FUNCTION_BLOCK EL3014
VAR
	_io : EL3xx4_Data;
	{attribute addProperty Name "WcState"}
	_wcState : WcStateInputToggle;
	{attribute addProperty Name "Info data"}
	_infoData : InfoDataAds;
END_VAR

PROPERTY IO : REFERENCE TO EL3xx4_Data
GET
IO REF= _io;
END_GET
END_PROPERTY

PROPERTY WcState : REFERENCE TO WcStateInputToggle
GET
WcState REF= _wcState;
END_GET
END_PROPERTY

END_FUNCTION_BLOCK

(* stored: Version 1.1.0.1, ProductVersion 3.1.4024.9
   POU EL3014: Id {15204826-2c94-02ae-383a-80dd5a00157f}, SpecialFunc None
   Property IO: Id {5d69b753-5e9f-0a8a-1825-ed3196d35c7d}
   Get Get: Id {15a7178a-8502-054c-059a-f62f5f305586}
   Property WcState: Id {3f8e7f82-eb6f-045c-2af1-5be9366a57f5}
   Get Get: Id {7f9673ac-4e59-0ccc-1138-c05592d45af6} *)
